// TIA Portal project "Operadores" (V16)

(* hardware
DEVICE "S7-1200 station_1"  S7-1200 Station
   slot 0: "Rack_0"  S7-1200 Rack  Rack  V1.0
   slot 1: "PLC_1"  CPU 1214C AC/DC/Rly  6ES7 214-1BG40-0XB0  V4.4
*)

// ===== PLC "PLC_1"  CPU 1214C AC/DC/Rly =====

VAR_GLOBAL   // PLC tag table "Tabla de variables estándar"
   "Tag_1" AT %I0.0 : Bool;
   "Tag_2" AT %I0.1 : Bool;
   "M_CONTA_ASC" AT %MW120 : Int;
   "Tag_3" AT %I0.4 : Bool;
   "Tag_4" AT %I0.5 : Bool;
   "M_CONTA_DESC" AT %MD101 : DWord;
   "Tag_5" AT %MW115 : Int;
   "Tag_6" AT %MW116 : Word;
   "Tag_7" AT %MW118 : Word;
   "Tag_8" AT %MW117 : Word;
   "Tag_9" AT %MW119 : Word;
END_VAR

// folder: System blocks/Program resources

DATA_BLOCK "IEC_Counter_0_DB"   // DB1
{ S7_Optimized_Access := 'TRUE' }
AUTHOR : Simatic
FAMILY : IEC
NAME : CNTR
VERSION : 1.0
// stored: InstanceOfName IEC_COUNTER
"IEC_COUNTER"
BEGIN
END_DATA_BLOCK

DATA_BLOCK "IEC_Counter_0_DB_1"   // DB2
{ S7_Optimized_Access := 'TRUE' }
AUTHOR : Simatic
FAMILY : IEC
NAME : CNTR
VERSION : 1.0
// stored: InstanceOfName IEC_COUNTER
"IEC_COUNTER"
BEGIN
END_DATA_BLOCK

// folder: (top level)

ORGANIZATION_BLOCK "Main"   // OB1, LAD, ProgramCycle
TITLE = "Main Program Sweep (Cycle)"
{ S7_Optimized_Access := 'TRUE' }
VERSION : 0.1
   VAR_INPUT
      Initial_Call : Bool;   // Initial call of this OB
      Remanence : Bool;   // =True, if remanent data are available
   END_VAR
BEGIN

REGION Network 1
   // CONTADORES
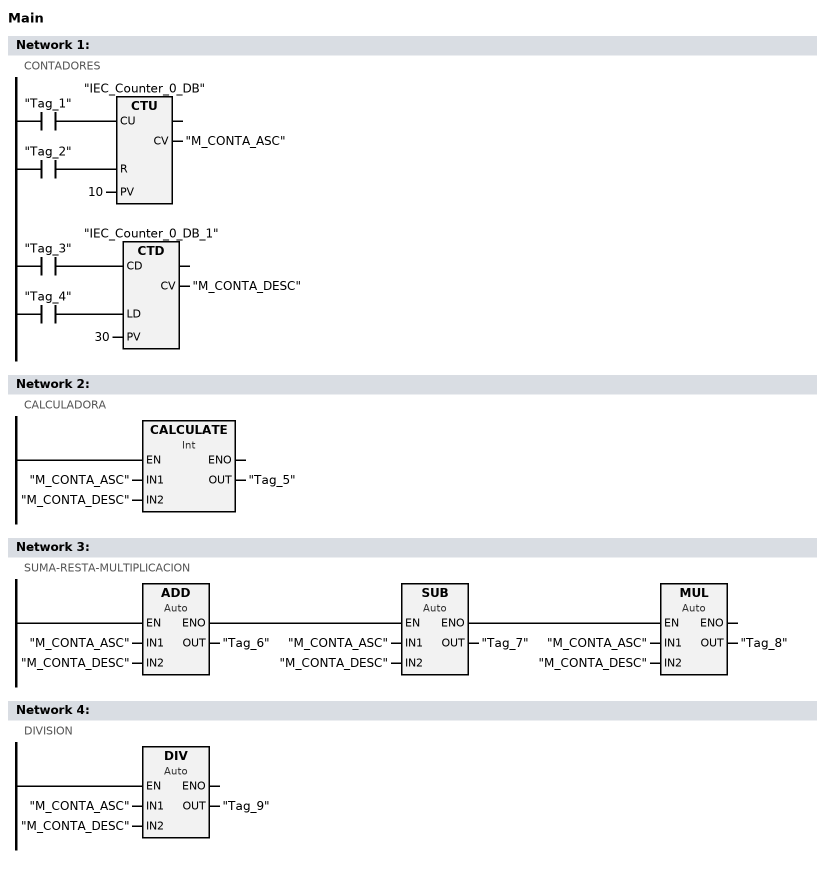
   "IEC_Counter_0_DB".CTU(CU := "Tag_1", R := "Tag_2", PV := 10, CV => "M_CONTA_ASC");
   "IEC_Counter_0_DB_1".CTD(CD := "Tag_3", LD := "Tag_4", PV := 30, CV => "M_CONTA_DESC");
END_REGION

REGION Network 2
   // CALCULADORA
   RUNG wire#powerrail
      { S7_Templates := "SrcType := Int"; S7_Expression := "IN1+IN2" } Calculate(in1 := "M_CONTA_ASC", in2 := "M_CONTA_DESC", out => "Tag_5")
   END_RUNG
   // the same network as SCL:
   "Tag_5" := "M_CONTA_ASC"+"M_CONTA_DESC";
END_REGION

REGION Network 3
   // SUMA-RESTA-MULTIPLICACION
   RUNG wire#powerrail
      Add(in1 := "M_CONTA_ASC", in2 := "M_CONTA_DESC", out => "Tag_6")
      Sub(in1 := "M_CONTA_ASC", in2 := "M_CONTA_DESC", out => "Tag_7")
      Mul(in1 := "M_CONTA_ASC", in2 := "M_CONTA_DESC", out => "Tag_8")
   END_RUNG
   // the same network as SCL:
   "Tag_6" := "M_CONTA_ASC" + "M_CONTA_DESC";
   "Tag_7" := "M_CONTA_ASC" - "M_CONTA_DESC";
   "Tag_8" := "M_CONTA_ASC" * "M_CONTA_DESC";
END_REGION

REGION Network 4
   // DIVISION
   RUNG wire#powerrail
      Div(in1 := "M_CONTA_ASC", in2 := "M_CONTA_DESC", out => "Tag_9")
   END_RUNG
   // the same network as SCL:
   "Tag_9" := "M_CONTA_ASC" / "M_CONTA_DESC";
END_REGION
END_ORGANIZATION_BLOCK